PROGRAM StewartTransform
VAR
END_VAR

METHOD PRIVATE xyz2zyx : ARRAY [0..2] OF REAL
VAR_INPUT
	phi : ARRAY [0..2] OF REAL;
END_VAR

VAR
	t1: REAL;
	t2: REAL;
	t3: REAL;
	t4: REAL;
	t5: REAL;
	t6: REAL;
	t7: REAL;
	t8: REAL;
END_VAR
// Maple optimized code
t1 := COS(phi[0]);
t2 := SIN(phi[1]);
t3 := SIN(phi[2]);
t4 := SIN(phi[0]);
t5 := COS(phi[2]);
t6 := t1 * t3;
t7 := t4 * t5;
t8 := COS(phi[1]);

xyz2zyx[0] := ATAN((t6 * t2 + t7)/(t1 * t8));
xyz2zyx[1] := -ASIN(-t1 * t2 * t5 + t3 * t4);
xyz2zyx[2] := ATAN((t7 * t2 + t6)/(t5 * t8));
END_METHOD

METHOD PRIVATE zyx2xyz : ARRAY [0..2] OF REAL
VAR_INPUT
	phi : ARRAY [0..2] OF REAL;
END_VAR

VAR
	t1: REAL;
	t2: REAL;
	t3: REAL;
	t4: REAL;
	t5: REAL;
	t6: REAL;
	t7: REAL;
	t8: REAL;
END_VAR
// Maple optimized code
t1 := SIN(phi[0]);
t2 := COS(phi[2]);
t3 := COS(phi[0]);
t4 := SIN(phi[1]);
t5 := SIN(phi[2]);
t6 := t3 * t5;
t7 := t1 * t2;
t8 := COS(phi[1]);

zyx2xyz[0] := ATAN((-t6 * t4 + t7)/(t3 * t8));
zyx2xyz[1] := ASIN(t3 * t4 * t2 + t1 * t5);
zyx2xyz[2] := ATAN((-t7 * t4 + t6)/( t2 * t8));
END_METHOD

END_PROGRAM

(* stored: Version 1.1.0.1, ProductVersion 3.1.4020.12
   POU StewartTransform: Id {b49d46a0-cf0b-47ca-9fd7-30991f5bfe9c}, SpecialFunc None
   Method xyz2zyx: Id {a99a340d-f442-470c-9732-27b8b5c20761}
   Method zyx2xyz: Id {dd6255de-a145-4cee-9644-ce2cf275d1dc} *)
